// Mitsubishi GX Works2 project: 14   PLC: FX3U/FX3UC

PROGRAM MAIN
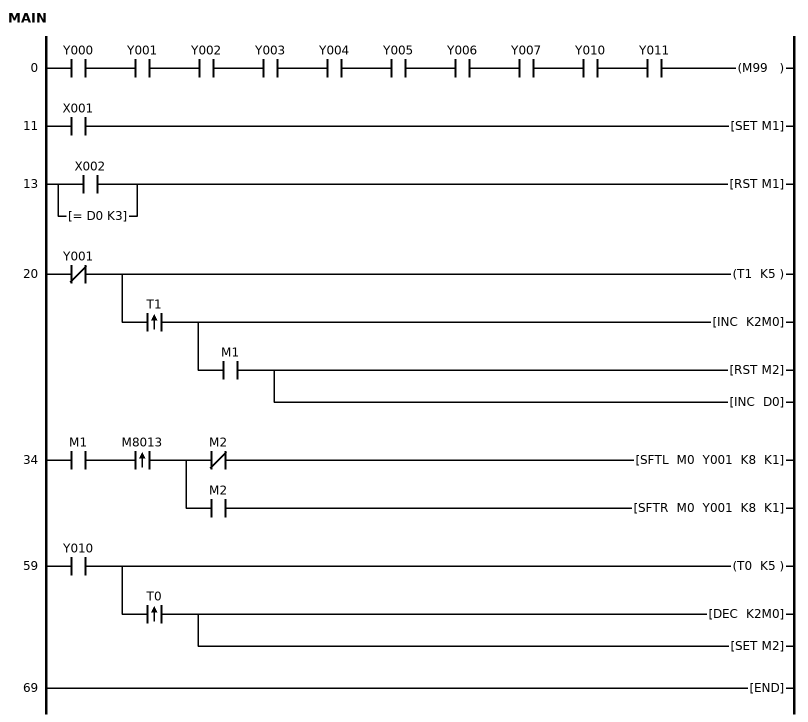
0     LD      Y000
      AND     Y001
      AND     Y002
      AND     Y003
      AND     Y004
      AND     Y005
      AND     Y006
      AND     Y007
      AND     Y010
      AND     Y011
      OUT     M99
11    LD      X001
      SET     M1
13    LD      X002
      OR=     D0 K3
      RST     M1
20    LDI     Y001
      OUT     T1 K5
      ANDP    T1
      INC     K2M0
      AND     M1
      RST     M2
      INC     D0
34    LD      M1
      ANDP    M8013
      MPS
      ANI     M2
      SFTL    M0 Y001 K8 K1
      MPP
      AND     M2
      SFTR    M0 Y001 K8 K1
59    LD      Y010
      OUT     T0 K5
      ANDP    T0
      DEC     K2M0
      SET     M2
69    END
END_PROGRAM
